% RSLogix 500 project Project_2.RSS, saved by version 8.30.00.16 %
PROJECT "UNTITLED"    % processor: Bul.1763 MicroLogix 1100 Series B %

PROGRAM FILES
  LAD 2 "MAIN"  3 rungs
  LAD 3 "CONTROL"  11 rungs
  LAD 4 "IO"  8 rungs

DATA FILES
  O0 OUTPUT  5 elements
  I1 INPUT  7 elements
  S2 STATUS  66 elements
  B3 BINARY  1 elements
  T4 TIMER  1 elements
  C5 COUNTER  1 elements
  R6 CONTROL  1 elements
  N7 INTEGER  3 elements
  F8 FLOAT  1 elements

LADDER 2 "MAIN"
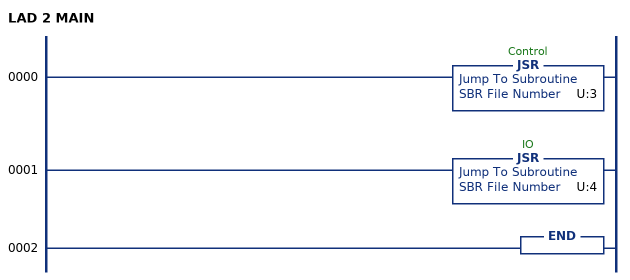
% Rung: 0 %
SOR JSR U:3 EOR
%   U:3  "Control" %
% Rung: 1 %
SOR JSR U:4 EOR
%   U:4  "IO" %
% Rung: 2 %
SOR END EOR

LADDER 3 "CONTROL"
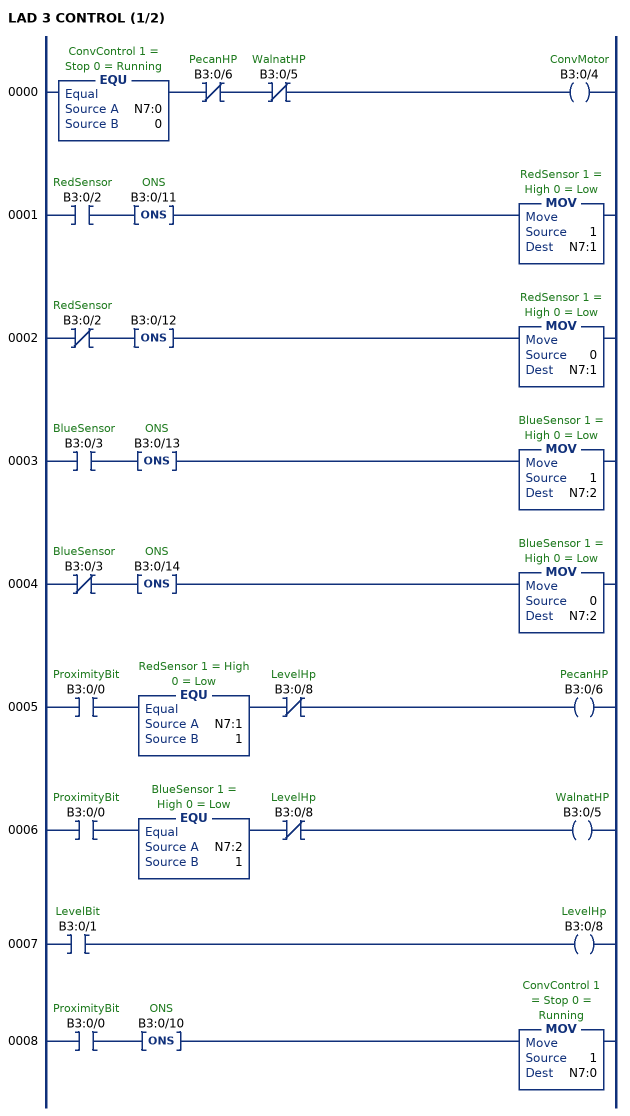
% Rung: 0 %
SOR EQU N7:0 0 XIO B3:0/6 XIO B3:0/5 OTE B3:0/4 EOR
%   N7:0  "ConvControl 1 = Stop 0 = Running" %
%   B3:0/6  "PecanHP" %
%   B3:0/5  "WalnatHP" %
%   B3:0/4  "ConvMotor" %
% Rung: 1 %
SOR XIC B3:0/2 ONS B3:0/11 MOV 1 N7:1 EOR
%   B3:0/2  "RedSensor" %
%   B3:0/11  "ONS" %
%   N7:1  "RedSensor 1 = High 0 = Low" %
% Rung: 2 %
SOR XIO B3:0/2 ONS B3:0/12 MOV 0 N7:1 EOR
%   B3:0/2  "RedSensor" %
%   N7:1  "RedSensor 1 = High 0 = Low" %
% Rung: 3 %
SOR XIC B3:0/3 ONS B3:0/13 MOV 1 N7:2 EOR
%   B3:0/3  "BlueSensor" %
%   B3:0/13  "ONS" %
%   N7:2  "BlueSensor 1 = High 0 = Low" %
% Rung: 4 %
SOR XIO B3:0/3 ONS B3:0/14 MOV 0 N7:2 EOR
%   B3:0/3  "BlueSensor" %
%   B3:0/14  "ONS" %
%   N7:2  "BlueSensor 1 = High 0 = Low" %
% Rung: 5 %
SOR XIC B3:0/0 EQU N7:1 1 XIO B3:0/8 OTE B3:0/6 EOR
%   B3:0/0  "ProximityBit" %
%   N7:1  "RedSensor 1 = High 0 = Low" %
%   B3:0/8  "LevelHp" %
%   B3:0/6  "PecanHP" %
% Rung: 6 %
SOR XIC B3:0/0 EQU N7:2 1 XIO B3:0/8 OTE B3:0/5 EOR
%   B3:0/0  "ProximityBit" %
%   N7:2  "BlueSensor 1 = High 0 = Low" %
%   B3:0/8  "LevelHp" %
%   B3:0/5  "WalnatHP" %
% Rung: 7 %
SOR XIC B3:0/1 OTE B3:0/8 EOR
%   B3:0/1  "LevelBit" %
%   B3:0/8  "LevelHp" %
% Rung: 8 %
SOR XIC B3:0/0 ONS B3:0/10 MOV 1 N7:0 EOR
%   B3:0/0  "ProximityBit" %
%   B3:0/10  "ONS" %
%   N7:0  "ConvControl 1 = Stop 0 = Running" %

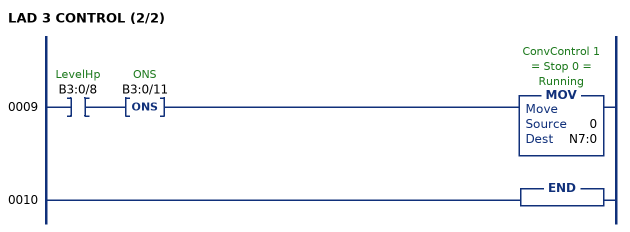
% Rung: 9 %
SOR XIC B3:0/8 ONS B3:0/11 MOV 0 N7:0 EOR
%   B3:0/8  "LevelHp" %
%   B3:0/11  "ONS" %
%   N7:0  "ConvControl 1 = Stop 0 = Running" %
% Rung: 10 %
SOR END EOR

LADDER 4 "IO"
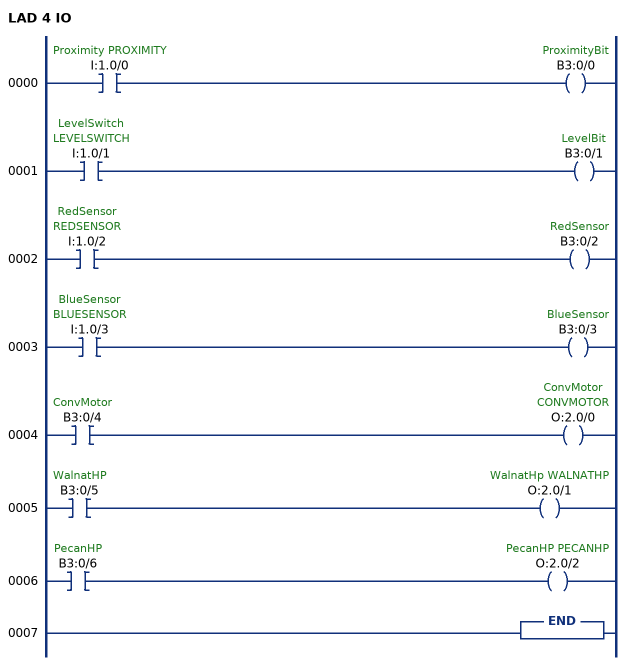
% Rung: 0 %
SOR XIC I:1.0/0 OTE B3:0/0 EOR
%   I:1.0/0  PROXIMITY  "Proximity" %
%   B3:0/0  "ProximityBit" %
% Rung: 1 %
SOR XIC I:1.0/1 OTE B3:0/1 EOR
%   I:1.0/1  LEVELSWITCH  "LevelSwitch" %
%   B3:0/1  "LevelBit" %
% Rung: 2 %
SOR XIC I:1.0/2 OTE B3:0/2 EOR
%   I:1.0/2  REDSENSOR  "RedSensor" %
%   B3:0/2  "RedSensor" %
% Rung: 3 %
SOR XIC I:1.0/3 OTE B3:0/3 EOR
%   I:1.0/3  BLUESENSOR  "BlueSensor" %
%   B3:0/3  "BlueSensor" %
% Rung: 4 %
SOR XIC B3:0/4 OTE O:2.0/0 EOR
%   B3:0/4  "ConvMotor" %
%   O:2.0/0  CONVMOTOR  "ConvMotor" %
% Rung: 5 %
SOR XIC B3:0/5 OTE O:2.0/1 EOR
%   B3:0/5  "WalnatHP" %
%   O:2.0/1  WALNATHP  "WalnatHp" %
% Rung: 6 %
SOR XIC B3:0/6 OTE O:2.0/2 EOR
%   B3:0/6  "PecanHP" %
%   O:2.0/2  PECANHP  "PecanHP" %
% Rung: 7 %
SOR END EOR

OTHER DOCUMENTED ADDRESSES
  B3:0/9  "ConvControl"
